FUNCTION F_CheckDivReal : REAL
VAR_INPUT
	divisor: REAL;
END_VAR

IF divisor = 0 THEN
	F_CheckDivReal:=1;
ELSE
	F_CheckDivReal:=divisor;
END_IF;

END_FUNCTION

(* stored: Version 1.1.0.1, ProductVersion 3.1.4022.6
   POU F_CheckDivReal: Id {00a4d3fc-2bda-4f08-8d66-495c27276c0e}, SpecialFunc None *)
